// TIA Portal V19 export
VAR_GLOBAL   // PLC tag table "DQ"
END_VAR
